(* Logix 5000 project; controller Machine_Maintenance_Lab2 vendor 1 type 14 code 155 rev 36.11; software revision 36.00 *)

TASK MainTask (continuous, watchdog 500 ms) : MainProgram

MODULES
   Local : vendor 1 type 14 code 155 (PointIO 0, rev 36.11)
      Discrete_IO : Embedded (PointIO 1, rev 36.11, Output RPI 20 ms)
END_MODULES

PROGRAM MainProgram   (* main routine MainRoutine *)
VAR
   counter : COUNTER;
   CycleCounter : COUNTER;
   delay : TIMER;
   HighCycleTimer : COUNTER;
   i_CycleDone : ALIAS FOR o_CycleDone;
   i_GreenPB : ALIAS FOR Local:1:I.Data.0;
   i_GreenPB_ConveyorStart : ALIAS FOR i_GreenPB;
   i_GreenPBLight_Conveyor1ON : ALIAS FOR o_GreenPBLight_Conveyor1ON;
   i_Pause : ALIAS FOR Pause;
   i_Piston : ALIAS FOR Local:1:O.Data.2;
   i_RedPB_StopButton : ALIAS FOR Local:1:I.Data.1;
   i_RedPBLight_Conveyor2ON : ALIAS FOR o_RedPBLight_Conveyor2ON;
   i_Turnkey : ALIAS FOR Local:1:I.Data.2;
   i_Turnkey_ItemSensor : ALIAS FOR i_Turnkey;
   ItemCounter1 : COUNTER;
   ItemCounterLeft : COUNTER;
   ItemCounterRight : COUNTER;
   LowCycleTimer : COUNTER;
   NewCycle : BOOL;
   o_CycleDone : BOOL;
   o_GreenPBLight : ALIAS FOR Local:1:O.Data.0;
   o_GreenPBLight_Conveyor1ON : ALIAS FOR o_GreenPBLight;
   o_Piston : ALIAS FOR i_Piston;
   o_RedPBLight : ALIAS FOR Local:1:O.Data.1;
   o_RedPBLight_Conveyor2ON : ALIAS FOR o_RedPBLight;
   o_YellowLate : ALIAS FOR Local:1:O.Data.2;
   OS_Out : BOOL;
   Pause : BOOL;
   ResetDelay : TIMER;
   RTO : TIMER;
   ThreeSecTimer : TIMER;
   timer : TIMER;
   TimerHighCycle : TIMER;
   TimerLowCycle : TIMER;
   TOF : TIMER;
   TON : TIMER;
   TurnkeyOneShot : BOOL;
END_VAR

ROUTINE MainRoutine   (* ladder *)
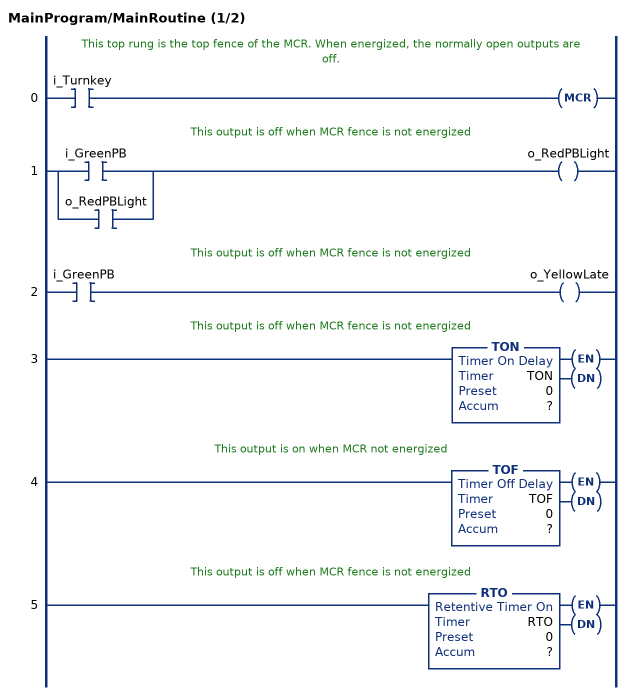
   // This top rung is the top fence of the MCR. When energized, the normally open outputs are off.
   0: XIC(i_Turnkey)MCR();
   // This output is off when MCR fence is not energized
   1: [XIC(i_GreenPB) ,XIC(o_RedPBLight) ]OTE(o_RedPBLight);
   // This output is off when MCR fence is not energized
   2: XIC(i_GreenPB)OTE(o_YellowLate);
   // This output is off when MCR fence is not energized
   3: TON(TON,?,?);
   // This output is on when MCR not energized
   4: TOF(TOF,?,?);
   // This output is off when MCR fence is not energized
   5: RTO(RTO,?,?);
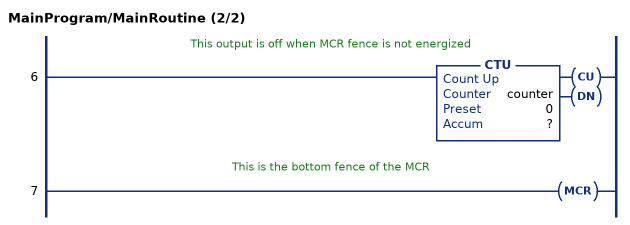
   // This output is off when MCR fence is not energized
   6: CTU(counter,?,?);
   // This is the bottom fence of the MCR
   7: MCR();
END_ROUTINE
END_PROGRAM
